PROGRAM MAIN
VAR
 	diKapSensor1 AT %I* : BOOL ;
 	diKapSensor2 AT %I* : BOOL ;
 
 	bMinneKapasativ1 : BOOL := 0 ;
	bMinneKapasativ2 : BOOL := 0 ;
 
END_VAR

bMinneKapasativ1 := diKapSensor1;
bMinneKapasativ2 := diKapSensor2;

END_PROGRAM

(* stored: Version 1.1.0.1, ProductVersion 3.1.4024.9
   POU MAIN: Id {d2bdd337-d709-463b-9776-8a15215056b6}, SpecialFunc None *)
